TYPE StepperENCControl :
STRUCT
	EnableLatchC : BOOL;
	EnableLatchPositiveEdge : BOOL;
	SetCounter : BOOL;
	EnableLatchNegativeEdge : BOOL;
	SetCounterValue : UDINT;
END_STRUCT
END_TYPE

(* stored: Version 1.1.0.1, ProductVersion 3.1.4024.9
   DUT StepperENCControl: Id {f0436a79-a568-4c0a-b1eb-93be32123967} *)
